INTERFACE I_LineBuilder EXTENDS T_QueryInterface

END_INTERFACE

(* stored: Version 1.1.0.1, ProductVersion 3.1.4024.4
   Itf I_LineBuilder: Id {25de0b71-969b-4988-a3f7-e3b24d80f633} *)
